(* CoDeSys 2.3.10.0 project: main.prx *)
(* Libraries: TcSystemBCxx50.lbx 11.2.10 15:45:50, TcBaseBCxx50.lbx 29.3.07 07:21:36, STANDARD.LBX 5.12.03 09:02:30 *)

(* Task configuration *)
TASK Standard (PRIORITY := 0, INTERVAL := T#20ms);
	MAIN
	ADS_init();
	led();
END_TASK
TASK sensors (PRIORITY := 1, INTERVAL := T#5ms);
	Prohibited_states();
	sensors();
END_TASK

(* Global variable list: Global_Variables *)
VAR_GLOBAL
	Ads_Udp_send_Stack : ARRAY [1..116] OF BOOL; (*информационный массив для передачи по ADS*)
	Ads_Udp_receive_Stack : ARRAY [1..116] OF BOOL; (*информационный массив для формирования*)
	Ads_Udp_old_received_Stack : ARRAY [1..116] OF BOOL; (*старый информационный массив для форсирования*)
	Ads_Udp_empty_Stack : ARRAY [1..116] OF BOOL;
	out_led AT %Q*:BOOL;
	udp_reset_alarm : BOOL := FALSE;
	in_button AT %I*:BOOL;

	led_blink	: BOOL:=FALSE;


	switch : BOOL;
	led_status:INT := 0;

	alarm_flag:BOOL := FALSE;
	reset_alarm:BOOL := FALSE;

	OPEN_POOL0 AT %Q*: BOOL;
	OPEN_POOL1 AT %Q*: BOOL;
	OPEN_1 AT %Q*: BOOL;
	OPEN_WC2_LIBRARY AT %Q*: BOOL;
	OPEN_WC_CHILDREN AT %Q*: BOOL;

	CLOSE_POOL0 AT %Q*: BOOL;
	CLOSE_POOL1 AT %Q*: BOOL;
	CLOSE_1 AT %Q*: BOOL;
	CLOSE_WC2_LIBRARY AT %Q*: BOOL;
	CLOSE_WC_CHILDREN AT %Q*: BOOL;

	SENSOR_INPUT1_1 AT %I*: BOOL;
	SENSOR_INPUT1_2 AT %I*: BOOL;
	SENSOR_INPUT1_3 AT %I*: BOOL;
	SENSOR_INPUT1_4 AT %I*: BOOL;
	SENSOR_INPUT1_5 AT %I*: BOOL;
	SENSOR_INPUT1_6 AT %I*: BOOL;
	SENSOR_INPUT1_7 AT %I*: BOOL;
	SENSOR_INPUT1_8 AT %I*: BOOL;
	SENSOR_INPUT1_9 AT %I*: BOOL;
	SENSOR_INPUT1_10 AT %I*: BOOL;
	SENSOR_INPUT1_11 AT %I*: BOOL;
	SENSOR_INPUT1_12 AT %I*: BOOL;
	SENSOR_INPUT1_13 AT %I*: BOOL;
	SENSOR_INPUT1_14 AT %I*: BOOL;
	SENSOR_INPUT1_15 AT %I*: BOOL;
	SENSOR_INPUT1_16 AT %I*: BOOL;

	SENSOR_INPUT2_1 AT %I*: BOOL;
	SENSOR_INPUT2_2 AT %I*: BOOL;
	SENSOR_INPUT2_3 AT %I*: BOOL;
	SENSOR_INPUT2_4 AT %I*: BOOL;
	SENSOR_INPUT2_5 AT %I*: BOOL;
	SENSOR_INPUT2_6 AT %I*: BOOL;
	SENSOR_INPUT2_7 AT %I*: BOOL;
	SENSOR_INPUT2_8 AT %I*: BOOL;
	SENSOR_INPUT2_9 AT %I*: BOOL;
	SENSOR_INPUT2_10 AT %I*: BOOL;
	SENSOR_INPUT2_11 AT %I*: BOOL;
	SENSOR_INPUT2_12 AT %I*: BOOL;
	SENSOR_INPUT2_13 AT %I*: BOOL;
	SENSOR_INPUT2_14 AT %I*: BOOL;
	SENSOR_INPUT2_15 AT %I*: BOOL;
	SENSOR_INPUT2_16 AT %I*: BOOL;
	SENSOR_INPUT2_17 AT %I*: BOOL;
	SENSOR_INPUT2_18 AT %I*: BOOL;
	SENSOR_INPUT2_19 AT %I*: BOOL;
	SENSOR_INPUT2_20 AT %I*: BOOL;
	SENSOR_INPUT2_21 AT %I*: BOOL;
	SENSOR_INPUT2_22 AT %I*: BOOL;
	SENSOR_INPUT2_23 AT %I*: BOOL;
	SENSOR_INPUT2_24 AT %I*: BOOL;
	SENSOR_INPUT2_25 AT %I*: BOOL;
	SENSOR_INPUT2_26 AT %I*: BOOL;		(*нет такого сенсора, физически между 25 и 27 подключена кнопка*)
	SENSOR_INPUT2_27 AT %I*: BOOL;
	SENSOR_INPUT2_28 AT %I*: BOOL;
	SENSOR_INPUT2_29 AT %I*: BOOL;
	SENSOR_INPUT2_30 AT %I*: BOOL;
	SENSOR_INPUT2_31 AT %I*: BOOL;
	SENSOR_INPUT2_32 AT %I*: BOOL;

	sensors_group_0_pool: BOOL;
	sensors_group_0_heater: BOOL;
	sensors_group_0_wc: BOOL;
	sensors_group_1: BOOL;
	sensors_group_2_lib_wc: BOOL;
	sensors_group_2_lv_wc: BOOL;
	sensors_group_2_children_wc: BOOL;
	sensors_group_undefined: BOOL;
	sensors_techrooms: BOOL;

	FLAG01_1: BOOL;
	FLAG01_2: BOOL;
	FLAG01_3: BOOL;
	FLAG01_4: BOOL;
	FLAG01_5: BOOL;
	FLAG01_6: BOOL;
	FLAG01_7: BOOL;
	FLAG01_8: BOOL;
	FLAG01_9: BOOL;
	FLAG01_10: BOOL;
	FLAG01_11: BOOL;
	FLAG01_12: BOOL;
	FLAG01_13: BOOL;
	FLAG01_14: BOOL;
	FLAG01_15: BOOL;
	FLAG01_16: BOOL;
	FLAG02_1: BOOL;
	FLAG02_2: BOOL;
	FLAG02_3: BOOL;
	FLAG02_4: BOOL;
	FLAG02_5: BOOL;
	FLAG02_6: BOOL;
	FLAG02_7: BOOL;
	FLAG02_8: BOOL;
	FLAG02_9: BOOL;
	FLAG02_10: BOOL;
	FLAG02_11: BOOL;
	FLAG02_12: BOOL;
	FLAG02_13: BOOL;
	FLAG02_14: BOOL;
	FLAG02_15: BOOL;
	FLAG02_16: BOOL;
	FLAG02_17: BOOL;
	FLAG02_18: BOOL;
	FLAG02_19: BOOL;
	FLAG02_20: BOOL;
	FLAG02_21: BOOL;
	FLAG02_22: BOOL;
	FLAG02_23: BOOL;
	FLAG02_24: BOOL;
	FLAG02_25: BOOL;
	FLAG02_26: BOOL;
	FLAG02_27: BOOL;
	FLAG02_28: BOOL;
	FLAG02_29: BOOL;
	FLAG02_30: BOOL;
	FLAG02_31: BOOL;
	FLAG02_32: BOOL;

END_VAR

(* Global variable list: TwinCAT_Configuration *)
(* Generated automatically by TwinCAT - (read only) *)
VAR_CONFIG
	.out_led AT %QX4.0 : BOOL;
	.in_button AT %IX8.0 : BOOL;
	.OPEN_POOL0 AT %QX0.1 : BOOL;
	.OPEN_POOL1 AT %QX0.2 : BOOL;
	.OPEN_1 AT %QX0.3 : BOOL;
	.OPEN_WC2_LIBRARY AT %QX0.4 : BOOL;
	.OPEN_WC_CHILDREN AT %QX0.5 : BOOL;
	.CLOSE_POOL0 AT %QX0.6 : BOOL;
	.CLOSE_POOL1 AT %QX0.7 : BOOL;
	.CLOSE_1 AT %QX1.0 : BOOL;
	.CLOSE_WC2_LIBRARY AT %QX1.1 : BOOL;
	.CLOSE_WC_CHILDREN AT %QX1.2 : BOOL;
	.SENSOR_INPUT1_1 AT %IX0.1 : BOOL;
	.SENSOR_INPUT1_2 AT %IX0.2 : BOOL;
	.SENSOR_INPUT1_3 AT %IX0.3 : BOOL;
	.SENSOR_INPUT1_4 AT %IX0.4 : BOOL;
	.SENSOR_INPUT1_5 AT %IX0.5 : BOOL;
	.SENSOR_INPUT1_6 AT %IX0.6 : BOOL;
	.SENSOR_INPUT1_7 AT %IX0.7 : BOOL;
	.SENSOR_INPUT1_8 AT %IX1.0 : BOOL;
	.SENSOR_INPUT1_9 AT %IX1.1 : BOOL;
	.SENSOR_INPUT1_10 AT %IX1.2 : BOOL;
	.SENSOR_INPUT1_11 AT %IX1.3 : BOOL;
	.SENSOR_INPUT1_12 AT %IX1.4 : BOOL;
	.SENSOR_INPUT1_13 AT %IX1.5 : BOOL;
	.SENSOR_INPUT1_14 AT %IX1.6 : BOOL;
	.SENSOR_INPUT1_15 AT %IX1.7 : BOOL;
	.SENSOR_INPUT1_16 AT %IX2.0 : BOOL;
	.SENSOR_INPUT2_1 AT %IX2.1 : BOOL;
	.SENSOR_INPUT2_2 AT %IX2.2 : BOOL;
	.SENSOR_INPUT2_3 AT %IX2.3 : BOOL;
	.SENSOR_INPUT2_4 AT %IX2.4 : BOOL;
	.SENSOR_INPUT2_5 AT %IX2.5 : BOOL;
	.SENSOR_INPUT2_6 AT %IX2.6 : BOOL;
	.SENSOR_INPUT2_7 AT %IX2.7 : BOOL;
	.SENSOR_INPUT2_8 AT %IX3.0 : BOOL;
	.SENSOR_INPUT2_9 AT %IX3.1 : BOOL;
	.SENSOR_INPUT2_10 AT %IX3.2 : BOOL;
	.SENSOR_INPUT2_11 AT %IX3.3 : BOOL;
	.SENSOR_INPUT2_12 AT %IX3.4 : BOOL;
	.SENSOR_INPUT2_13 AT %IX3.5 : BOOL;
	.SENSOR_INPUT2_14 AT %IX3.6 : BOOL;
	.SENSOR_INPUT2_15 AT %IX3.7 : BOOL;
	.SENSOR_INPUT2_16 AT %IX4.0 : BOOL;
	.SENSOR_INPUT2_17 AT %IX4.1 : BOOL;
	.SENSOR_INPUT2_18 AT %IX4.2 : BOOL;
	.SENSOR_INPUT2_19 AT %IX4.3 : BOOL;
	.SENSOR_INPUT2_20 AT %IX4.4 : BOOL;
	.SENSOR_INPUT2_21 AT %IX4.5 : BOOL;
	.SENSOR_INPUT2_22 AT %IX4.6 : BOOL;
	.SENSOR_INPUT2_23 AT %IX4.7 : BOOL;
	.SENSOR_INPUT2_24 AT %IX5.0 : BOOL;
	.SENSOR_INPUT2_25 AT %IX5.1 : BOOL;
	.SENSOR_INPUT2_26 AT %IX5.2 : BOOL;
	.SENSOR_INPUT2_27 AT %IX5.3 : BOOL;
	.SENSOR_INPUT2_28 AT %IX5.4 : BOOL;
	.SENSOR_INPUT2_29 AT %IX5.5 : BOOL;
	.SENSOR_INPUT2_30 AT %IX5.6 : BOOL;
	.SENSOR_INPUT2_31 AT %IX5.7 : BOOL;
	.SENSOR_INPUT2_32 AT %IX6.0 : BOOL;
END_VAR

(* POU MAIN, ST *)
PROGRAM MAIN
VAR

	in_button_state:BOOL;
	Alarm: 	INT;
	First : BOOL := TRUE;
	mb_: BOOL;

	Falling_edge_trig : F_TRIG;
	ALARM_sup: BOOL;
END_VAR
IF(First = TRUE) THEN
		OPEN_POOL0 := TRUE;
		OPEN_POOL1 := TRUE;
		OPEN_1 := TRUE;
		OPEN_WC2_LIBRARY := TRUE;
		OPEN_WC_CHILDREN := TRUE;
		CLOSE_POOL0 := FALSE;
		CLOSE_POOL1 := FALSE;
		CLOSE_1 := FALSE;
		CLOSE_WC2_LIBRARY := FALSE;
		CLOSE_WC_CHILDREN := FALSE;
First := FALSE;
END_IF;

IF(in_button = 0) THEN
	in_button_state := 0;
END_IF;

IF (in_button_state = 0 AND in_button > 0 AND NOT(alarm_flag)) THEN
	switch := NOT(switch);
	in_button_state := 1;
END_IF;

IF(reset_alarm OR udp_reset_alarm) THEN
	alarm_flag := FALSE;
	switch := FALSE;
END_IF;

IF(alarm_flag) THEN
	led_blink:=TRUE;
ELSE
	led_blink:=FALSE;
END_IF;

(*если нажата кнопка, то все вкл. или все выкл.*)
	IF(switch) THEN

		CLOSE_POOL0 := TRUE;
		CLOSE_POOL1 := TRUE;
		CLOSE_1:= TRUE;
		CLOSE_WC2_LIBRARY := TRUE;
		CLOSE_WC_CHILDREN := TRUE;

		OPEN_POOL0 := FALSE;
		OPEN_POOL1 := FALSE;
		OPEN_1 := FALSE;
		OPEN_WC2_LIBRARY := FALSE;
		OPEN_WC_CHILDREN := FALSE;
ELSE

		IF(sensors_group_0_pool) THEN
			OPEN_POOL1:=FALSE;
			CLOSE_POOL1:=TRUE;
		END_IF;

		IF(sensors_group_0_wc) THEN
			OPEN_POOL0:=FALSE;
			CLOSE_POOL0:=TRUE;
		END_IF;

		IF(sensors_group_1 OR sensors_group_0_heater) THEN
			OPEN_1:=FALSE;
			CLOSE_1:=TRUE;
		END_IF;

		IF(sensors_group_2_lib_wc OR sensors_group_2_lv_wc) THEN
			OPEN_WC2_LIBRARY:=FALSE;
			CLOSE_WC2_LIBRARY:=TRUE;
		END_IF;

		IF(sensors_group_2_children_wc) THEN
			OPEN_WC_CHILDREN:=FALSE;
			CLOSE_WC_CHILDREN:=TRUE;
		END_IF;

		IF(sensors_group_undefined OR sensors_techrooms) THEN
			OPEN_POOL1:=FALSE;
			CLOSE_POOL1:=TRUE;
			OPEN_POOL0:=FALSE;
			CLOSE_POOL0:=TRUE;
			OPEN_1:=FALSE;
			CLOSE_1:=TRUE;
			OPEN_WC2_LIBRARY:=FALSE;
			CLOSE_WC2_LIBRARY:=TRUE;
			OPEN_WC_CHILDREN:=FALSE;
			CLOSE_WC_CHILDREN:=TRUE;
		END_IF;


	(*Если была сработка хотя бы одного датчика, то выходим из текущего шага*)
		IF(sensors_group_0_pool OR sensors_group_0_heater OR sensors_group_0_wc OR sensors_group_1 OR
                        sensors_group_2_lib_wc OR sensors_group_2_lv_wc OR sensors_group_2_children_wc OR sensors_group_undefined OR sensors_techrooms) THEN
			alarm_flag:=TRUE;
			RETURN;
		END_IF;

Falling_edge_trig (CLK := alarm_flag, Q => );
IF ((reset_alarm OR udp_reset_alarm OR in_button_state) AND NOT(alarm_flag)) THEN
		OPEN_POOL0 := TRUE;
		OPEN_POOL1 := TRUE;
		OPEN_1 := TRUE;
		OPEN_WC2_LIBRARY := TRUE;
		OPEN_WC_CHILDREN := TRUE;
		CLOSE_POOL0 := FALSE;
		CLOSE_POOL1 := FALSE;
		CLOSE_1 := FALSE;
		CLOSE_WC2_LIBRARY := FALSE;
		CLOSE_WC_CHILDREN := FALSE;
		ALARM_sup := FALSE;
END_IF;
END_IF;
END_PROGRAM

(* POU ADS_init, ST *)
PROGRAM ADS_init
VAR
	First: BOOL := TRUE;
	k: INT;
	Rec_Not_Empty: BOOL;
END_VAR
(*ads stack init*)
	Ads_Udp_send_Stack[1] := SENSOR_INPUT1_1;
	Ads_Udp_send_Stack[2] := SENSOR_INPUT1_2;
	Ads_Udp_send_Stack[3] := SENSOR_INPUT1_3;
	Ads_Udp_send_Stack[4] := SENSOR_INPUT1_4;
	Ads_Udp_send_Stack[5] := SENSOR_INPUT1_5;
	Ads_Udp_send_Stack[6] := SENSOR_INPUT1_6;
	Ads_Udp_send_Stack[7] := SENSOR_INPUT1_7;
	Ads_Udp_send_Stack[8] := SENSOR_INPUT1_8;
	Ads_Udp_send_Stack[9] := SENSOR_INPUT1_9;
	Ads_Udp_send_Stack[10] := SENSOR_INPUT1_10;
	Ads_Udp_send_Stack[11] := SENSOR_INPUT1_11;
	Ads_Udp_send_Stack[12] := SENSOR_INPUT1_12;
	Ads_Udp_send_Stack[13] := SENSOR_INPUT1_13;
	Ads_Udp_send_Stack[14] := SENSOR_INPUT1_14;
	Ads_Udp_send_Stack[15] := SENSOR_INPUT1_15;
	Ads_Udp_send_Stack[16] := SENSOR_INPUT1_16;
	Ads_Udp_send_Stack[17] := SENSOR_INPUT2_1;
	Ads_Udp_send_Stack[18] := SENSOR_INPUT2_2;
	Ads_Udp_send_Stack[19] := SENSOR_INPUT2_3;
	Ads_Udp_send_Stack[20] := SENSOR_INPUT2_4;
	Ads_Udp_send_Stack[21] := SENSOR_INPUT2_5;
	Ads_Udp_send_Stack[22] := SENSOR_INPUT2_6;
	Ads_Udp_send_Stack[23] := SENSOR_INPUT2_7;
	Ads_Udp_send_Stack[24] := SENSOR_INPUT2_8;
	Ads_Udp_send_Stack[25] := SENSOR_INPUT2_9;
	Ads_Udp_send_Stack[26] := SENSOR_INPUT2_10;
	Ads_Udp_send_Stack[27] := SENSOR_INPUT2_11;
	Ads_Udp_send_Stack[28] := SENSOR_INPUT2_12;
	Ads_Udp_send_Stack[29] := SENSOR_INPUT2_13;
	Ads_Udp_send_Stack[30] := SENSOR_INPUT2_14;
	Ads_Udp_send_Stack[31] := SENSOR_INPUT2_15;
	Ads_Udp_send_Stack[32] := SENSOR_INPUT2_16;
	Ads_Udp_send_Stack[33] := SENSOR_INPUT2_17;
	Ads_Udp_send_Stack[34] := SENSOR_INPUT2_18;
	Ads_Udp_send_Stack[35] := SENSOR_INPUT2_19;
	Ads_Udp_send_Stack[36] := SENSOR_INPUT2_20;
	Ads_Udp_send_Stack[37] := SENSOR_INPUT2_21;
	Ads_Udp_send_Stack[38] := SENSOR_INPUT2_22;
	Ads_Udp_send_Stack[39] := SENSOR_INPUT2_23;
	Ads_Udp_send_Stack[40] := SENSOR_INPUT2_24;
	Ads_Udp_send_Stack[41] := SENSOR_INPUT2_25;
	Ads_Udp_send_Stack[42] := SENSOR_INPUT2_26;
	Ads_Udp_send_Stack[43] := SENSOR_INPUT2_27;
	Ads_Udp_send_Stack[44] := SENSOR_INPUT2_28;
	Ads_Udp_send_Stack[45] := SENSOR_INPUT2_29;
	Ads_Udp_send_Stack[46] := SENSOR_INPUT2_30;
	Ads_Udp_send_Stack[47] := SENSOR_INPUT2_31;
	Ads_Udp_send_Stack[48] := SENSOR_INPUT2_32;
	Ads_Udp_send_Stack[49] := sensors_group_0_pool;
	Ads_Udp_send_Stack[50] := sensors_group_0_wc;
	Ads_Udp_send_Stack[51] := sensors_group_1;
	Ads_Udp_send_Stack[52] := sensors_group_2_lib_wc;
	Ads_Udp_send_Stack[53] := sensors_group_2_lv_wc;
	Ads_Udp_send_Stack[54] := sensors_group_2_children_wc;
	Ads_Udp_send_Stack[55] := OPEN_POOL0;
	Ads_Udp_send_Stack[56] := OPEN_POOL1;
	Ads_Udp_send_Stack[57] := OPEN_1;
	Ads_Udp_send_Stack[58] := OPEN_WC2_LIBRARY;
	Ads_Udp_send_Stack[59] := OPEN_WC_CHILDREN;
	Ads_Udp_send_Stack[60] := CLOSE_POOL0;
	Ads_Udp_send_Stack[61] := CLOSE_POOL1;
	Ads_Udp_send_Stack[62] := CLOSE_1;
	Ads_Udp_send_Stack[63] := CLOSE_WC2_LIBRARY;
	Ads_Udp_send_Stack[64] := CLOSE_WC_CHILDREN;
	Ads_Udp_send_Stack[65] := alarm_flag;
	Ads_Udp_send_Stack[66] := udp_reset_alarm;
(*расширение протокола*)
	Ads_Udp_send_Stack[67] := sensors_group_0_heater;
	Ads_Udp_send_Stack[68] := sensors_group_undefined;
	Ads_Udp_send_Stack[69] := FLAG01_1;
	Ads_Udp_send_Stack[70] := FLAG01_2;
	Ads_Udp_send_Stack[71] := FLAG01_3;
	Ads_Udp_send_Stack[72] := FLAG01_4;
	Ads_Udp_send_Stack[73] := FLAG01_5;
	Ads_Udp_send_Stack[74] := FLAG01_6;
	Ads_Udp_send_Stack[75] := FLAG01_7;
	Ads_Udp_send_Stack[76] := FLAG01_8;
	Ads_Udp_send_Stack[77] := FLAG01_9;
	Ads_Udp_send_Stack[78] := FLAG01_10;
	Ads_Udp_send_Stack[79] := FLAG01_11;
	Ads_Udp_send_Stack[80] := FLAG01_12;
	Ads_Udp_send_Stack[81] := FLAG01_13;
	Ads_Udp_send_Stack[82] := FLAG01_14;
	Ads_Udp_send_Stack[83] := FLAG01_15;
	Ads_Udp_send_Stack[84] := FLAG01_16;
	Ads_Udp_send_Stack[85] := FLAG02_1;
	Ads_Udp_send_Stack[86] := FLAG02_2;
	Ads_Udp_send_Stack[87] := FLAG02_3;
	Ads_Udp_send_Stack[88] := FLAG02_4;
	Ads_Udp_send_Stack[89] := FLAG02_5;
	Ads_Udp_send_Stack[90] := FLAG02_6;
	Ads_Udp_send_Stack[91] := FLAG02_7;
	Ads_Udp_send_Stack[92] := FLAG02_8;
	Ads_Udp_send_Stack[93] := FLAG02_9;
	Ads_Udp_send_Stack[94] := FLAG02_10;
	Ads_Udp_send_Stack[95] := FLAG02_11;
	Ads_Udp_send_Stack[96] := FLAG02_12;
	Ads_Udp_send_Stack[97] := FLAG02_13;
	Ads_Udp_send_Stack[98] := FLAG02_14;
	Ads_Udp_send_Stack[99] := FLAG02_15;
	Ads_Udp_send_Stack[100] := FLAG02_16;
	Ads_Udp_send_Stack[101] := FLAG02_17;
	Ads_Udp_send_Stack[102] := FLAG02_18;
	Ads_Udp_send_Stack[103] := FLAG02_19;
	Ads_Udp_send_Stack[104] := FLAG02_20;
	Ads_Udp_send_Stack[105] := FLAG02_21;
	Ads_Udp_send_Stack[106] := FLAG02_22;
	Ads_Udp_send_Stack[107] := FLAG02_23;
	Ads_Udp_send_Stack[108] := FLAG02_24;
	Ads_Udp_send_Stack[109] := FLAG02_25;
	Ads_Udp_send_Stack[110] := FLAG02_26;
	Ads_Udp_send_Stack[111] := FLAG02_27;
	Ads_Udp_send_Stack[112] := FLAG02_28;
	Ads_Udp_send_Stack[113] := FLAG02_29;
	Ads_Udp_send_Stack[114] := FLAG02_30;
	Ads_Udp_send_Stack[115] := FLAG02_31;
	Ads_Udp_send_Stack[116] := FLAG02_32;
	ADS_block;

Rec_Not_Empty := FALSE;
FOR k := 1 TO 116 DO
IF (Ads_Udp_receive_Stack[k] = Ads_Udp_empty_Stack[k]) THEN
Rec_Not_Empty := (Rec_Not_Empty OR FALSE);
ELSE
Rec_Not_Empty := (Rec_Not_Empty OR TRUE);
END_IF;
END_FOR;

IF(Rec_Not_Empty) THEN
IF(First = TRUE) THEN
Ads_Udp_old_received_Stack := Ads_Udp_receive_Stack;
First := FALSE;
END_IF;

	udp_reset_alarm := Ads_Udp_receive_Stack[66];
IF(Ads_Udp_receive_Stack[55] = NOT(Ads_Udp_old_received_Stack[55] ) OR Ads_Udp_receive_Stack[60] = NOT(Ads_Udp_old_received_Stack[60] )) THEN
	OPEN_POOL0 := Ads_Udp_receive_Stack[55];
	CLOSE_POOL0 := Ads_Udp_receive_Stack[60];
	Ads_Udp_send_Stack[55] := Ads_Udp_receive_Stack[55];
	Ads_Udp_send_Stack[60] := Ads_Udp_receive_Stack[60];
END_IF;
IF(Ads_Udp_receive_Stack[56] = NOT(Ads_Udp_old_received_Stack[56] ) OR Ads_Udp_receive_Stack[61] = NOT(Ads_Udp_old_received_Stack[61] )) THEN
	OPEN_POOL1 := Ads_Udp_receive_Stack[56];
	CLOSE_POOL1 := Ads_Udp_receive_Stack[61];
	Ads_Udp_send_Stack[56] := Ads_Udp_receive_Stack[56];
	Ads_Udp_send_Stack[61] := Ads_Udp_receive_Stack[61];
END_IF;
IF(Ads_Udp_receive_Stack[57] = NOT(Ads_Udp_old_received_Stack[57] ) OR Ads_Udp_receive_Stack[62] = NOT(Ads_Udp_old_received_Stack[62] )) THEN
	OPEN_1 := Ads_Udp_receive_Stack[57];
	CLOSE_1 := Ads_Udp_receive_Stack[62];
	Ads_Udp_send_Stack[57] := Ads_Udp_receive_Stack[57];
	Ads_Udp_send_Stack[62] := Ads_Udp_receive_Stack[62];
END_IF;
IF(Ads_Udp_receive_Stack[58] = NOT(Ads_Udp_old_received_Stack[58] ) OR Ads_Udp_receive_Stack[63] = NOT(Ads_Udp_old_received_Stack[63] )) THEN
	OPEN_WC2_LIBRARY := Ads_Udp_receive_Stack[58];
	CLOSE_WC2_LIBRARY := Ads_Udp_receive_Stack[63];
	Ads_Udp_send_Stack[58] := Ads_Udp_receive_Stack[58];
	Ads_Udp_send_Stack[63] := Ads_Udp_receive_Stack[63];
END_IF;
IF(Ads_Udp_receive_Stack[59] = NOT(Ads_Udp_old_received_Stack[59] ) OR Ads_Udp_receive_Stack[64] = NOT(Ads_Udp_old_received_Stack[64] )) THEN
	OPEN_WC_CHILDREN := Ads_Udp_receive_Stack[59];
	CLOSE_WC_CHILDREN := Ads_Udp_receive_Stack[64];
	Ads_Udp_send_Stack[59] := Ads_Udp_receive_Stack[59];
	Ads_Udp_send_Stack[64] := Ads_Udp_receive_Stack[64];
END_IF;

IF (Ads_Udp_send_Stack[65] = FALSE AND Ads_Udp_receive_Stack[66] = TRUE) THEN Ads_Udp_receive_Stack[66] := FALSE; Ads_Udp_send_Stack[66] := FALSE; END_IF;

	FLAG01_1:= Ads_Udp_receive_Stack[69];
	FLAG01_2 := Ads_Udp_receive_Stack[70];
	FLAG01_3 := Ads_Udp_receive_Stack[71];
	FLAG01_4 := Ads_Udp_receive_Stack[72];
	FLAG01_5 := Ads_Udp_receive_Stack[73];
	FLAG01_6 := Ads_Udp_receive_Stack[74];
	FLAG01_7 := Ads_Udp_receive_Stack[75];
	FLAG01_8 := Ads_Udp_receive_Stack[76];
	FLAG01_9 := Ads_Udp_receive_Stack[77];
	FLAG01_10 := Ads_Udp_receive_Stack[78];
	FLAG01_11 := Ads_Udp_receive_Stack[79];
	FLAG01_12 := Ads_Udp_receive_Stack[80];
	FLAG01_13 := Ads_Udp_receive_Stack[81];
	FLAG01_14 := Ads_Udp_receive_Stack[82];
	FLAG01_15 := Ads_Udp_receive_Stack[83];
	FLAG01_16 := Ads_Udp_receive_Stack[84];
	FLAG02_1 := Ads_Udp_receive_Stack[85];
	FLAG02_2 := Ads_Udp_receive_Stack[86];
	FLAG02_3 := Ads_Udp_receive_Stack[87];
	FLAG02_4 := Ads_Udp_receive_Stack[88];
	FLAG02_5 := Ads_Udp_receive_Stack[89];
	FLAG02_6 := Ads_Udp_receive_Stack[90];
	FLAG02_7 := Ads_Udp_receive_Stack[91];
	FLAG02_8 := Ads_Udp_receive_Stack[92];
	FLAG02_9 := Ads_Udp_receive_Stack[93];
	FLAG02_10 := Ads_Udp_receive_Stack[94];
	FLAG02_11 := Ads_Udp_receive_Stack[95];
	FLAG02_12 := Ads_Udp_receive_Stack[96];
	FLAG02_13 := Ads_Udp_receive_Stack[97];
	FLAG02_14 := Ads_Udp_receive_Stack[98];
	FLAG02_15 := Ads_Udp_receive_Stack[99];
	FLAG02_16 := Ads_Udp_receive_Stack[100];
	FLAG02_17 := Ads_Udp_receive_Stack[101];
	FLAG02_18 := Ads_Udp_receive_Stack[102];
	FLAG02_19 := Ads_Udp_receive_Stack[103];
	FLAG02_20 := Ads_Udp_receive_Stack[104];
	FLAG02_21 := Ads_Udp_receive_Stack[105];
	FLAG02_22 := Ads_Udp_receive_Stack[106];
	FLAG02_23 := Ads_Udp_receive_Stack[107];
	FLAG02_24 := Ads_Udp_receive_Stack[108];
	FLAG02_25 := Ads_Udp_receive_Stack[109];
	FLAG02_26 := Ads_Udp_receive_Stack[110];
	FLAG02_27 := Ads_Udp_receive_Stack[111];
	FLAG02_28 := Ads_Udp_receive_Stack[112];
	FLAG02_29 := Ads_Udp_receive_Stack[113];
	FLAG02_30 := Ads_Udp_receive_Stack[114];
	FLAG02_31 := Ads_Udp_receive_Stack[115];
	FLAG02_32 := Ads_Udp_receive_Stack[116];

Ads_Udp_old_received_Stack := Ads_Udp_receive_Stack;
END_IF;
END_PROGRAM

(* POU ADS_block, CFC *)
PROGRAM ADS_block
VAR
	Repeater1: TON;
	ADSwritecxbc: ADSWRITE;
	ADSreadcxbc: ADSREAD;
	First: BOOL := TRUE;
END_VAR
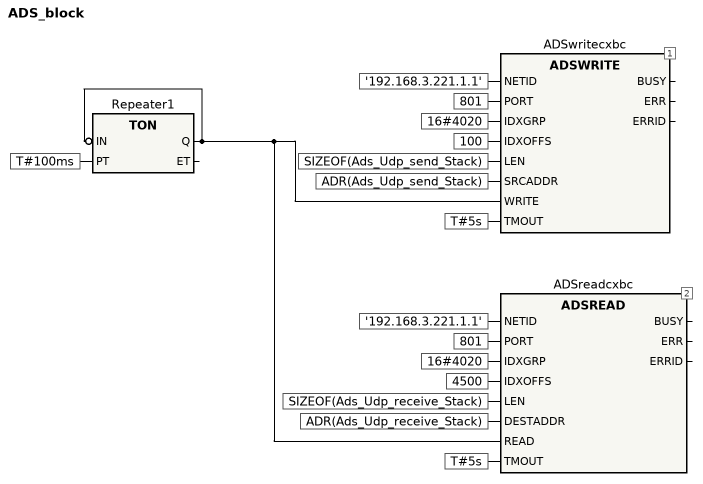
_CFC_ (* Continuous Function Chart, elements in execution order *)
#0 Repeater1:TON(IN: NOT #0.Q, PT: T#100ms)
#1 ADSwritecxbc:ADSWRITE(NETID: '192.168.3.221.1.1', PORT: 801, IDXGRP: 16#4020, IDXOFFS: 100, LEN: SIZEOF(Ads_Udp_send_Stack), SRCADDR: ADR(Ads_Udp_send_Stack), WRITE: #0.Q, TMOUT: T#5s)
#2 ADSreadcxbc:ADSREAD(NETID: '192.168.3.221.1.1', PORT: 801, IDXGRP: 16#4020, IDXOFFS: 4500, LEN: SIZEOF(Ads_Udp_receive_Stack), DESTADDR: ADR(Ads_Udp_receive_Stack), READ: #0.Q, TMOUT: T#5s)
_END_CFC_
(* the same logic as Structured Text *)
Repeater1(IN := NOT Repeater1.Q, PT := T#100ms);
ADSwritecxbc(NETID := '192.168.3.221.1.1', PORT := 801, IDXGRP := 16#4020, IDXOFFS := 100, LEN := SIZEOF(Ads_Udp_send_Stack), SRCADDR := ADR(Ads_Udp_send_Stack), WRITE := Repeater1.Q, TMOUT := T#5s);
ADSreadcxbc(NETID := '192.168.3.221.1.1', PORT := 801, IDXGRP := 16#4020, IDXOFFS := 4500, LEN := SIZEOF(Ads_Udp_receive_Stack), DESTADDR := ADR(Ads_Udp_receive_Stack), READ := Repeater1.Q, TMOUT := T#5s);
END_PROGRAM

(* POU led, CFC *)
PROGRAM led
VAR
	Timer1: TON;
	Timer2: TOF;
	timer_in: TON;
END_VAR
VAR (* helpers for the ST form of the networks *)
	_t4 : BOOL;
	_t20 : BOOL;
END_VAR
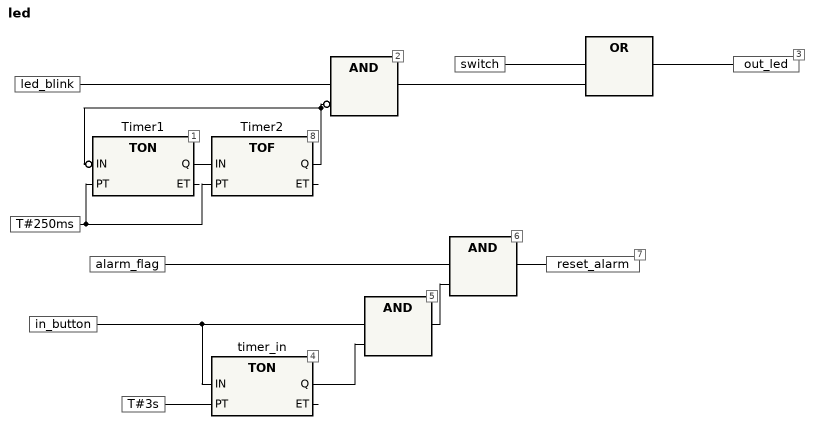
_CFC_ (* Continuous Function Chart, elements in execution order *)
#0 OR(switch, #2)
#1 Timer1:TON(IN: NOT #8.Q, PT: T#250ms)
#2 AND(led_blink, NOT #8.Q)
#3 out_led <= #0
#4 timer_in:TON(IN: in_button, PT: T#3s)
#5 AND(in_button, #4.Q)
#6 AND(alarm_flag, #5)
#7 reset_alarm <= #6
#8 Timer2:TOF(IN: #1.Q, PT: T#250ms)
_END_CFC_
(* the same logic as Structured Text *)
_t20 := switch OR _t4;
Timer1(IN := NOT Timer2.Q, PT := T#250ms);
_t4 := led_blink AND NOT Timer2.Q;
out_led := _t20;
timer_in(IN := in_button, PT := T#3s);
reset_alarm := alarm_flag AND (in_button AND timer_in.Q);
Timer2(IN := Timer1.Q, PT := T#250ms);
END_PROGRAM

(* POU Prohibited_states, ST *)
PROGRAM Prohibited_states
VAR
END_VAR
IF(OPEN_POOL0 AND CLOSE_POOL0) THEN
OPEN_POOL0 := FALSE;
CLOSE_POOL0 := FALSE;
END_IF;
IF(OPEN_POOL1 AND CLOSE_POOL1) THEN
OPEN_POOL1 := FALSE;
CLOSE_POOL1 := FALSE;
END_IF;
IF(OPEN_1 AND CLOSE_1) THEN
OPEN_1 := FALSE;
CLOSE_1 := FALSE;
END_IF;
IF(OPEN_WC2_LIBRARY AND CLOSE_WC2_LIBRARY) THEN
OPEN_WC2_LIBRARY := FALSE;
CLOSE_WC2_LIBRARY := FALSE;
END_IF;
IF(OPEN_WC_CHILDREN AND CLOSE_WC_CHILDREN) THEN
OPEN_WC_CHILDREN := FALSE;
CLOSE_WC_CHILDREN := FALSE;
END_IF;
END_PROGRAM

(* POU sensors, ST *)
PROGRAM sensors
VAR
END_VAR
IF( SENSOR_INPUT2_27 AND NOT(FLAG02_27) OR		(*кнопка *)
     SENSOR_INPUT1_6 AND NOT(FLAG01_6) OR
     SENSOR_INPUT1_7 AND NOT(FLAG01_7) OR
     SENSOR_INPUT1_8 AND NOT(FLAG01_8) OR
     SENSOR_INPUT1_9 AND NOT(FLAG01_9) OR
     SENSOR_INPUT1_2 AND NOT(FLAG01_2) OR 			(*сигнал от Ajax на POOL_1*)									(**)
     SENSOR_INPUT1_10 AND NOT(FLAG01_10)) THEN		(*бескорпусной датчик в коридоре цоколь *)

		sensors_group_0_pool := TRUE;
ELSE
		sensors_group_0_pool := FALSE;
END_IF;


(* wc цоколь*)
IF(   SENSOR_INPUT2_27 AND NOT(FLAG02_27) OR		(*кнопка *)
	SENSOR_INPUT2_3 AND NOT(FLAG02_3) OR		(*датчик постирочной под раковиной*)
	SENSOR_INPUT1_11 AND NOT(FLAG01_11) OR		(*датчик под вентустановкой*)
	SENSOR_INPUT1_3 AND NOT(FLAG01_3) OR
	SENSOR_INPUT1_4 AND NOT(FLAG01_4) OR
	SENSOR_INPUT1_5 AND NOT(FLAG01_5) OR
	SENSOR_INPUT1_16 AND NOT(FLAG01_16) OR 		(*сигнал от Ajax на POOL_0*)										(**)
	SENSOR_INPUT2_2 AND NOT(FLAG02_2)) THEN		(*бескорпусной датчик в коридоре цоколь *)

		sensors_group_0_wc := TRUE;
ELSE
		sensors_group_0_wc := FALSE;
END_IF;

(*2й этаж -детская wc*)
IF(   SENSOR_INPUT2_21 AND NOT(FLAG02_21) OR
	SENSOR_INPUT2_32 AND NOT(FLAG02_32) OR 		(*сигнал от Ajax на WC_CHILDREN*)							(**)
	SENSOR_INPUT2_22 AND NOT(FLAG02_22)) THEN

		sensors_group_2_children_wc:= TRUE;
ELSE
		sensors_group_2_children_wc := FALSE;
END_IF;


(*2й этаж -библиотека*)
IF(   SENSOR_INPUT2_29 AND NOT(FLAG02_29) OR			(*кнопка *)
	SENSOR_INPUT2_14 AND NOT(FLAG02_14) OR
	SENSOR_INPUT2_25 AND NOT(FLAG02_25) OR 			(*сигнал от Ajax на WC_LIB*)									(**)
	SENSOR_INPUT2_16 AND NOT(FLAG02_16)) THEN

		sensors_group_2_lib_wc := TRUE;
ELSE
		sensors_group_2_lib_wc := FALSE;
END_IF;


(* санузел, хозяйская спальня*)
IF(SENSOR_INPUT2_29 AND NOT(FLAG02_29) OR			(*кнопка *)
	SENSOR_INPUT2_18 AND NOT(FLAG02_18) OR
	SENSOR_INPUT2_19 AND NOT(FLAG02_19) OR
	SENSOR_INPUT2_20 AND NOT(FLAG02_20)) THEN

		sensors_group_2_lv_wc := TRUE;
ELSE
		sensors_group_2_lv_wc := FALSE;
END_IF;

IF(SENSOR_INPUT1_1 AND NOT(FLAG01_1)  OR
	SENSOR_INPUT2_15 AND NOT(FLAG02_15) OR			(*датчик кухня кинозала *)
	SENSOR_INPUT1_15 AND NOT(FLAG01_15)) THEN		(*датчик теплового пункта в коридоре цоколь *)

		sensors_group_0_heater := TRUE;
ELSE
		sensors_group_0_heater := FALSE;
END_IF

IF(SENSOR_INPUT2_28 AND NOT(FLAG02_28) OR			(*кнопка *)
	SENSOR_INPUT2_24 AND NOT(FLAG02_24) OR 			(*сигнал от Ajax на 1ST FLOOR*)								(**)
	SENSOR_INPUT2_11 AND NOT(FLAG02_11)) THEN		(*датчик в кладовой 1-ый этаж (недоступен?) *)

		sensors_group_1 := TRUE;
ELSE
		sensors_group_1 := FALSE;
END_IF;

(*не работающие/заблокированные датчики*)
IF(
	SENSOR_INPUT1_12 AND NOT(FLAG01_12) OR
	SENSOR_INPUT1_13 AND NOT(FLAG01_13) OR
	SENSOR_INPUT2_4 AND NOT(FLAG02_4) OR
	SENSOR_INPUT2_5 AND NOT(FLAG02_5) OR
	SENSOR_INPUT2_6 AND NOT(FLAG02_6) OR
	SENSOR_INPUT2_7 AND NOT(FLAG02_7) OR
	SENSOR_INPUT2_8 AND NOT(FLAG02_8) OR
	SENSOR_INPUT2_9 AND NOT(FLAG02_9) OR
	SENSOR_INPUT2_10 AND NOT(FLAG02_10) OR
	SENSOR_INPUT2_12 AND NOT(FLAG02_12) OR
	SENSOR_INPUT2_13 AND NOT(FLAG02_13) OR
	SENSOR_INPUT2_17 AND NOT(FLAG02_17) OR
	SENSOR_INPUT2_23 AND NOT(FLAG02_23) OR
(*	SENSOR_INPUT2_26 AND NOT(FLAG02_26) OR 		нет такого сенсора, физически между 25 и 27 подключена кнопка*)
(*	SENSOR_INPUT2_27 AND NOT(FLAG02_27) OR
	SENSOR_INPUT2_28 AND NOT(FLAG02_28) OR
	SENSOR_INPUT2_29 AND NOT(FLAG02_29) OR             кнопки  *)
	SENSOR_INPUT2_30 AND NOT(FLAG02_30) OR
	SENSOR_INPUT2_31 AND NOT(FLAG02_31)) THEN

		sensors_group_undefined := TRUE;
ELSE
		sensors_group_undefined := FALSE;
END_IF;

IF(	SENSOR_INPUT1_14 AND NOT(FLAG01_14) OR           (*датчики протечек в щитовой 2_1 и серверной 1_14*)
	SENSOR_INPUT2_1 AND NOT(FLAG02_1)) THEN
		sensors_techrooms := TRUE;
ELSE
		sensors_techrooms := FALSE;
END_IF;
END_PROGRAM
